ABB RobotStudio station: Get_picture_legos_20180418-103907.rsstn

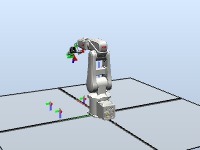
Station Get_picture_legos (saved by RobotStudio 6.6.7701.1025)
Controller System3
  mechanical unit ROB_1: IRB120_3_58__01, 6 joints, base frame (0, 0, 0) mm
Layout (positions relative to the parent item):
  - IRB120_3_58__01 [mechanism, from Robots\IRB120_3_58_G_01.rslib] at (0, 0, 0) mm; joint values [0, 0, 0, 0, 0.5236, 0] (rad or m)
  - MoveToViewpoint_2 [smart component, from Components\MoveToViewpoint.rslib]
      properties: Viewpoint=Viewpoint_4; Time=0
  - Camera_2 [smart component, from Components\Camera.rslib] at (0, 0, 0) mm
      properties: Path=D:\Produkt- og Designpsykologi\8. Semester\2. Robot Vision\Workshops; File Name=test
  - lego2x2_blue_2 [part] at (500, 0, 0) mm, rotated rx 90 ry 0 rz 0 deg
  - lego2x2_white_2 [part] at (-300, 0, 0) mm, rotated rx 90 ry 0 rz 0 deg
  - lego2x2_yellow_2 [part] at (0, 400, 0) mm, rotated rx 90 ry 0 rz 0 deg
  - Group_1 [graphiccomponentgroup]
  - SmartComponent_1 [smart component, from Libraries\SCHINK_WSG_GRIPPER.rslib] at (364.35, 0, 594) mm, rotated rx 180 ry 60 rz 180 deg
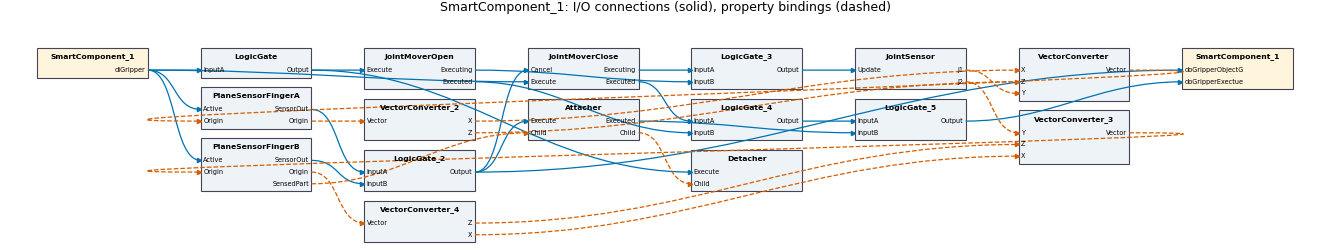
      connections:
        SmartComponent_1.diGripper -> LogicGate.InputA
        SmartComponent_1.diGripper -> PlaneSensorFingerA.Active
        SmartComponent_1.diGripper -> PlaneSensorFingerB.Active
        PlaneSensorFingerA.SensorOut -> LogicGate_2.InputA
        PlaneSensorFingerB.SensorOut -> LogicGate_2.InputB
        LogicGate_2.Output -> JointMoverClose.Cancel
        LogicGate_2.Output -> SmartComponent_1.doGripperObjectGrasped
        SmartComponent_1.diGripper -> JointMoverClose.Execute
        LogicGate.Output -> JointMoverOpen.Execute
        JointMoverClose.Executing -> LogicGate_3.InputA
        JointMoverOpen.Executing -> LogicGate_3.InputB
        LogicGate_3.Output -> JointSensor.Update
        LogicGate_2.Output -> Attacher.Execute
        LogicGate.Output -> Detacher.Execute
        JointMoverClose.Executed -> LogicGate_4.InputA
        JointMoverOpen.Executed -> LogicGate_4.InputB
        LogicGate_4.Output -> LogicGate_5.InputA
        Attacher.Executed -> LogicGate_5.InputB
        LogicGate_5.Output -> SmartComponent_1.doGripperExectued
        VectorConverter_2.X => VectorConverter.X
        VectorConverter_2.Z => VectorConverter.Z
        JointSensor.J1 => VectorConverter.Y
        PlaneSensorFingerA.Origin => VectorConverter_2.Vector
        VectorConverter.Vector => PlaneSensorFingerA.Origin
        JointSensor.J2 => VectorConverter_3.Y
        VectorConverter_4.Z => VectorConverter_3.Z
        VectorConverter_4.X => VectorConverter_3.X
        PlaneSensorFingerB.Origin => VectorConverter_4.Vector
        VectorConverter_3.Vector => PlaneSensorFingerB.Origin
        PlaneSensorFingerB.SensedPart => Attacher.Child
        Attacher.Child => Detacher.Child
    - SCHINK_WSG_GRIPPER [mechanism, from Libraries\SCHINK_WSG_GRIPPER.rslib] at (0, 0, 0) mm; joint values [0.0535, -0.0535] (rad or m)
    - PlaneSensorFingerA [smart component, from Components\PlaneSensor.rslib]
        properties: Origin=[-0.015 0.0535 0.13582]; Axis1=[0.03 0 0]; Axis2=[0 0 0.099]; SensedPart=(none)
      - _sensorPart_ [part, from Libraries\SCHINK_WSG_GRIPPER.rslib]
    - PlaneSensorFingerB [smart component, from Components\PlaneSensor.rslib]
        properties: Origin=[-0.015 -0.0535 0.13582]; Axis1=[0.03 0 0]; Axis2=[0 0 0.099]; SensedPart=(none)
      - _sensorPart_ [part, from Libraries\SCHINK_WSG_GRIPPER.rslib]
    - JointMoverClose [smart component, from Components\JointMover.rslib]
        properties: Mechanism=SCHINK_WSG_GRIPPER; Relative=false; Duration=2; J1=0; J2=0
    - JointMoverOpen [smart component, from Components\JointMover.rslib]
        properties: Mechanism=SCHINK_WSG_GRIPPER; Relative=false; Duration=2; J1=0.0535; J2=-0.0535
    - LogicGate [smart component, from Components\LogicGate.rslib]
        properties: Operator=NOT; Delay=0
    - LogicGate_2 [smart component, from Components\LogicGate.rslib]
        properties: Operator=AND; Delay=0
    - JointSensor [smart component, from Components\JointSensor.rslib]
        properties: Mechanism=SCHINK_WSG_GRIPPER; J1=0.0535; J2=-0.0535
    - LogicGate_3 [smart component, from Components\LogicGate.rslib]
        properties: Operator=OR; Delay=0
    - VectorConverter [smart component, from Components\VectorConverter.rslib]
        properties: X=-0.015; Y=0.0535; Z=0.13582; Vector=[-0.015 0.0535 0.13582]
    - VectorConverter_2 [smart component, from Components\VectorConverter.rslib]
        properties: X=-0.015; Y=0.0535; Z=0.13582; Vector=[-0.015 0.0535 0.13582]
    - VectorConverter_3 [smart component, from Components\VectorConverter.rslib]
        properties: X=-0.015; Y=-0.0535; Z=0.13582; Vector=[-0.015 -0.0535 0.13582]
    - VectorConverter_4 [smart component, from Components\VectorConverter.rslib]
        properties: X=-0.015; Y=-0.0535; Z=0.13582; Vector=[-0.015 -0.0535 0.13582]
    - Attacher [smart component, from Components\Attacher.rslib]
        properties: Parent=SCHINK_WSG_GRIPPER; Flange=0; Child=(none); Mount=false; Offset=[0 0 0]; Orientation=[0 0 0]
    - Detacher [smart component, from Components\Detacher.rslib]
        properties: Child=(none); KeepPosition=true
    - LogicGate_4 [smart component, from Components\LogicGate.rslib]
        properties: Operator=OR; Delay=0
    - LogicGate_5 [smart component, from Components\LogicGate.rslib]
        properties: Operator=OR; Delay=0
  - Pixel Points [part]
Attachment: Camera_2 is attached to IRB120_3_58__01 / Link6
Attachment: MoveToViewpoint_2 is attached to IRB120_3_58__01 / Base
Attachment: SmartComponent_1 is attached to IRB120_3_58__01 / Link6
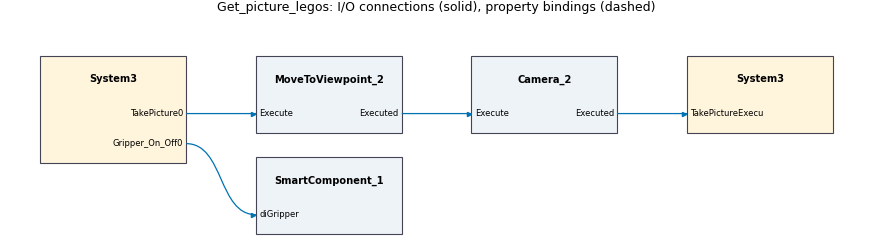
Station logic (signal -> signal, property => property):
  MoveToViewpoint_2.Executed -> Camera_2.Execute
  System3.TakePicture0 -> MoveToViewpoint_2.Execute
  Camera_2.Executed -> System3.TakePictureExecuted0
  System3.Gripper_On_Off0 -> SmartComponent_1.diGripper
Targets, tools, work objects and paths stored in the station, written as RAPID:
! task T_ROB1
MODULE FunctionHandler
  PERS tooldata defaultTool:=[TRUE,[[0,0,0],[1,0,0,0]],[1,[0,0,0.001],[1,0,0,0],0,0,0]];
  PERS wobjdata defaultWobj:=[FALSE,TRUE,"",[[0,0,0],[1,0,0,0]],[[0,0,0],[1,0,0,0]]];
  VAR signaldo defaultTakePictureActivationIO;
  VAR signaldi defaultTakePictureExecutedIO;
  PROC FH_TakePicture()
    SetDO defaultTakePictureActivationIO,1;
    WaitDI defaultTakePictureExecutedIO,1;
    SetDO defaultTakePictureActivationIO,0;
  ENDPROC
ENDMODULE

! task T_ROB1
MODULE CommandHandler
  PROC COMH_CommandListener()
  ENDPROC
ENDMODULE

! task T_ROB1
MODULE Module1
  CONST robtarget Target_10:=[[230.468,300,7.94],[0,0,1,0],[0,0,0,0],[9E+09,9E+09,9E+09,9E+09,9E+09,9E+09]];
  CONST robtarget Target_20:=[[480,300,10.171],[0,0,1,0],[0,0,0,2],[9E+09,9E+09,9E+09,9E+09,9E+09,9E+09]];
  CONST robtarget Target_30:=[[480,-77.629,7.886],[0,0,1,0],[-1,0,-1,0],[9E+09,9E+09,9E+09,9E+09,9E+09,9E+09]];
  PROC main()
    IP_Initialize;
    COMH_CommandListener;
  ENDPROC
ENDMODULE

! task T_ROB1
MODULE InitParameters
  PROC IP_Initialize()
    ConfL \Off;
    ConfJ \Off;
  ENDPROC
ENDMODULE

! task T_ROB1
MODULE CalibData
  PERS tooldata MyTool:=[TRUE,[[31.792631019,0,229.638935148],[0.945518576,0,0.325568154,0]],[1,[0,0,1],[1,0,0,0],0,0,0]];
  PERS tooldata SCHINK_WSG_GRIPPER_TOOL:=[TRUE,[[0,0,234.82],[1,0,0,0]],[5,[0,0,100],[1,0,0,0],0,0,0]];
ENDMODULE

